TYPE T_CodePRODUCEDATE : STRING[14];
END_TYPE

(* stored: Version 1.1.0.1
   DUT T_CodePRODUCEDATE: Id {dcec1c16-1f94-44b3-8175-fd09a8b95ab2} *)
